PROGRAM Service_sim
//---------------------------------Acutators simulation----------------------------------//
VAR
	TON_0: TON;
	TON_1: TON;
	TON_2: TON;
	TON_3: TON;
	TON_4: TON;
END_VAR

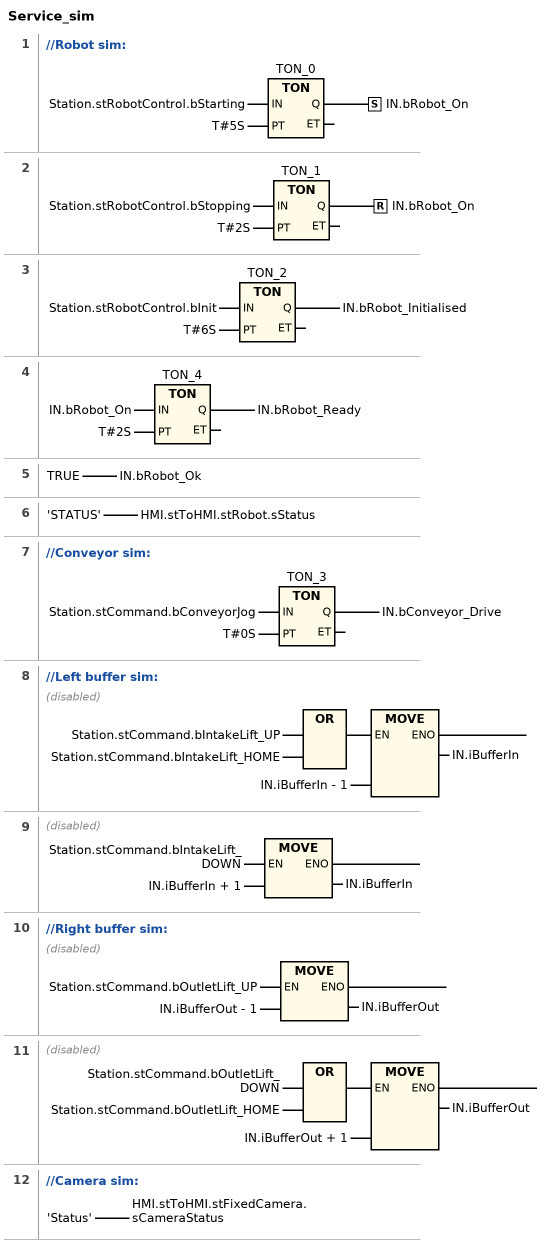
// NETWORK 1
// label: //Robot sim
TON_0(IN := Station.stRobotControl.bStarting, PT := T#5S); // TON
IN.bRobot_On S= TON_0.Q;

// NETWORK 2
TON_1(IN := Station.stRobotControl.bStopping, PT := T#2S); // TON
IN.bRobot_On R= TON_1.Q;

// NETWORK 3
TON_2(IN := Station.stRobotControl.bInit, PT := T#6S); // TON
IN.bRobot_Initialised := TON_2.Q;

// NETWORK 4
TON_4(IN := IN.bRobot_On, PT := T#2S); // TON
IN.bRobot_Ready := TON_4.Q;

// NETWORK 5
IN.bRobot_Ok := TRUE;

// NETWORK 6
HMI.stToHMI.stRobot.sStatus := 'STATUS';

// NETWORK 7
// label: //Conveyor sim
TON_3(IN := Station.stCommand.bConveyorJog, PT := T#0S); // TON
IN.bConveyor_Drive := TON_3.Q;

// NETWORK 8 (disabled)
// label: //Left buffer sim
// IF Station.stCommand.bIntakeLift_UP OR Station.stCommand.bIntakeLift_HOME THEN
//     IN.iBufferIn := IN.iBufferIn - 1;
// END_IF

// NETWORK 9 (disabled)
// IF Station.stCommand.bIntakeLift_DOWN THEN IN.iBufferIn := IN.iBufferIn + 1; END_IF

// NETWORK 10 (disabled)
// label: //Right buffer sim
// IF Station.stCommand.bOutletLift_UP THEN IN.iBufferOut := IN.iBufferOut - 1; END_IF

// NETWORK 11 (disabled)
// IF Station.stCommand.bOutletLift_DOWN OR Station.stCommand.bOutletLift_HOME THEN
//     IN.iBufferOut := IN.iBufferOut + 1;
// END_IF

// NETWORK 12
// label: //Camera sim
HMI.stToHMI.stFixedCamera.sCameraStatus := 'Status';

END_PROGRAM

(* stored: Version 1.1.0.1
   POU Service_sim: Id {01fa9ed5-c1a4-48cb-8090-d9aa32fd5f05}, SpecialFunc None *)
